{attribute 'qualified_only'}
{attribute 'strict'}
TYPE E_LeakLocation :
(
	NO_LEAK := 0,
	LOC1 := 1,
	LOC2 := 2,
	LOC3 := 4,
	LOC4 := 8,
	LOC5 := 16,
	LOC6 := 32
) BYTE;
END_TYPE

(* stored: Version 1.1.0.1, ProductVersion 3.1.4024.6
   DUT E_LeakLocation: Id {2f6f5662-e0e9-45ea-b191-3cdfc221cc16} *)
